(* PLC project Tc2_MC2_Camming.MC_SetCamOnlineChangeMode Demo, tc3-libraries-kb TwinCAT 3.1 *)
(* stored: creationDateTime 2026-05-21T00:00:00, modificationDateTime 2026-05-21T00:00:00 *)

PROGRAM P_Demo_MC_SetCamOnlineChangeMode
  VAR
    fbConfigCamActivation : MC_SetCamOnlineChangeMode;
    stChangeModeOpts : ST_SetOnlineChangeModeOptions;
    eActivationMode : MC_CamActivationMode;
    eMasterScaling : MC_CamScalingMode;
    eSlaveScaling : MC_CamScalingMode;
    lrSwitchOverMasterPos : LREAL := 0.0;
    nActiveCamId : MC_CAM_ID;
    bConfigureNow : BOOL := FALSE;
    rtConfigTrig : R_TRIG;
    bConfigDone : BOOL;
    bConfigBusy : BOOL;
    bConfigError : BOOL;
    nConfigErrorID : UDINT;
  END_VAR

// =============================================================================
// 场景：包装机系统初始化阶段 — 在 PLC 启动且完成 MC_CamTableSelect 加载
//       生产凸轮表后，配置该表的"在线修改激活策略"：未来用
//       MC_WriteMotionFunction* 写 cam 形状时，新数据排队等主轴回到 0 位
//       (lrSwitchOverMasterPos = 0.0) 才切换。这样跑产品过程中下发配方
//       不会在产品中段引起从轴跳变。
// 价值：把"写数据"和"激活时机"解耦 — 后续写 cam 的逻辑不再需要每次
//       判断"现在切安不安全"；NC 内核根据本配置以微秒级时序自动切换。
//       这是 cam runtime API 安全使用的核心机制。
// 验证步骤：
//   1) 编译登录；nActiveCamId 已由 MC_CamTableSelect 准备好。
//   2) eActivationMode 在 PLC 初始化时设为 MC_CAMACTIVATION_ATMASTERCAMPOS
//      （或工艺要求的其他枚举值，由项目算法填）；本例代码不显式赋值，
//      由调用方按需在线写入或在外部初始化代码中设置。
//   3) 在线 bConfigureNow := TRUE → R_TRIG 上升沿触发 Execute；
//      bConfigBusy 立 TRUE，1-N 周期后 bConfigDone := TRUE。
//   4) 此时本 FB 不会让任何 cam 形状变化 — 这是正常的（配置类 FB）。
//   5) 验证生效：随后调用 MC_WriteMotionFunctionPoint 修改某节点，
//      bWriteDone 后 watch Axis.Status.CamDataQueued — 应为 TRUE
//      (说明数据排队中)；主轴运动到 lrSwitchOverMasterPos = 0 时
//      CamDataQueued 变 FALSE，从轴轨迹切到新 cam。
//   6) 故障路径：nActiveCamId 传 0 或一个无效 ID 触发，应观察
//      bConfigError := TRUE。
// =============================================================================
// 说明：eActivationMode / eMasterScaling / eSlaveScaling 在本例为局部变
//       量，工程里通常在初始化段或配方表里赋值。本例不显式硬编码具体
//       枚举值（避免与 PDF 枚举定义脱节）。

rtConfigTrig(CLK := bConfigureNow);

// 单次完整调用：注意 ActivationPosition 是"未缩放"位置参考；
// 若应用层位置已经过 MasterScaling 缩放，调用前需先 / MasterScaling 反推。
fbConfigCamActivation(
    Execute            := rtConfigTrig.Q,
    ActivationMode     := eActivationMode,
    ActivationPosition := lrSwitchOverMasterPos,
    MasterScalingMode  := eMasterScaling,
    SlaveScalingMode   := eSlaveScaling,
    CamTableID         := nActiveCamId,
    Options            := stChangeModeOpts,
    Done               => bConfigDone,
    Busy               => bConfigBusy,
    Error              => bConfigError,
    ErrorID            => nConfigErrorID
);
END_PROGRAM
